{attribute addProperty BoxType "EL6080-0000-0018"}
{attribute addProperty Id "StatusAT %I*Status_8B1CA2AE1620InputsEMPTY_STRUCTURE000ControlAT %Q*Control_734938A41620OutputsEMPTY_STRUCTURE000WcStateAT %I*WcState_98A4DF7520.250InfoDataAT %I*InfoData_BC63D37F80100"}
{attribute addProperty CRC "3110452621"}
{attribute addProperty SizeInBites "114"}
{attribute addProperty SizeInBytes "14.25"}
TYPE EL6080_B3418C28 :
STRUCT
	{attribute addProperty Name "Status"}
	Status : Status_8B1CA2AE;
	{attribute addProperty Name "Inputs"}
	Inputs : EMPTY_STRUCTURE;
	{attribute addProperty Name "Control"}
	Control : Control_734938A4;
	{attribute addProperty Name "Outputs"}
	Outputs : EMPTY_STRUCTURE;
	{attribute addProperty Name "WcState"}
	WcState : WcState_98A4DF75;
	{attribute addProperty Name "InfoData"}
	InfoData : InfoData_BC63D37F;
END_STRUCT
END_TYPE

(* stored: Version 1.2.0.0, ProductVersion 3.1.4024.9
   DUT EL6080_B3418C28: Id {4b0475b2-73cb-4720-951e-24484ea1b9a7} *)
